VAR_GLOBAL
	bOn				AT%I*:		BOOL:= TRUE;
	bEMStop			AT%I*:		BOOL:= TRUE;
	bDoorsOk		AT%I*:		BOOL:= TRUE;
	bFuse			AT%I*:		BOOL:= TRUE;
END_VAR

(* stored: Version 1.1.0.1
   GVL IO: Id {fda10e4f-669f-010f-06b9-810ead0cb8ac} *)
